(* Logix 5000 project; controller CLASE_1 Emulate 5570 rev 28.11; software revision 28.02; part 6 of 15 *)
(* tags used below, declared in another part *)
   Inp_RunFdbk : BOOL;   // Input Signal: RUN feedback from motor
   Inp_PermOK : BOOL;   // 1=Permissives OK, motor can start
   Inp_NBPermOK : BOOL;   // 1=Non-Bypassable Permissives OK, motor can start
   Inp_IntlkOK : BOOL;   // 1=Interlocks OK, motor can start/run
   Inp_NBIntlkOK : BOOL;   // 1=Non-Bypassable Interlocks OK, motor can start/run
   Inp_IOFault : BOOL;   // Input Communication Status 0=OK, 1=fail
   Inp_Sim : BOOL;   // 1=Simulate working motor; 0=Start/Stop/ Monitor actual motor
   Inp_OvrdCmd : DINT;   // Override Mode Command: 0=None, 1=Stop, 2=Start
   Cfg_HasRunFdbk : BOOL;   // 1=Motor provides run feedback
   Cfg_UseRunFdbk : BOOL;   // 1=Motor run feedback should be used for failure checking
   Cfg_AllowLocal : BOOL;   // 1=Allow Local Start/Stop without alarm, 0=Start/Stop from HMI/prog only
   Cfg_PCmdClear : ALIAS FOR Mode.Cfg_PCmdClear;
   Cfg_OperStopPrio : BOOL;   // 1=OCmd_Stop available in any mode, 0=OCmd_Stop only in Oper, Maint modes.
   Cfg_OCmdResets : BOOL;   // 1=New Oper motor cmd. resets fault, 0=reset req'd to clear fault
   Cfg_ShedOnFailToStart : BOOL;   // 1=Stop Motor and Alarm on Fail to Start; 0=Alarm only on Fail to Start
   Cfg_ShedOnIOFault : BOOL;   // 1=Stop Motor and Alarm on I/O Fault; 0=Alarm only on I/O Fault
   PCmd_Start : BOOL;   // Program Command to Start Motor
   PCmd_Stop : BOOL;   // Program Command to Stop Motor
   OCmd_Start : BOOL;   // Operator Command to Start Motor
   OCmd_Stop : BOOL;   // Operator Command to Stop Motor
   Out_Run : BOOL;   // 1=Run Motor, 0=Stop Motor
   Out_Start : BOOL;   // 1=Start Motor, 0=Motor left in current state
   Out_Stop : BOOL;   // 1=Stop Motor, 0=Motor left in current state
   SrcQ_IO : SINT;   // Source and Quality of primary I/O (enumeration)
   SrcQ : SINT;   // Source and Quality of primary Val/Sts (enumeration)
   Val_Cmd : SINT;   // Device Command 0=None, 1=Stop, 2=Start
   Val_Sts : SINT;   // Device Confirmed Sts 0=? 1=Stopped, 2=Running, 7=Stopping, 8=Starting, 33=Disabled
   Val_Fault : SINT;   // Device Fault Status 0=None, 16=Fail to Start, 17 = Fail to Stop, 32=I/O Fault, 34=Config Error
   Val_Notify : SINT;   // Current Alarm Level and Acknowledgement (enumeration)
   Sts_Stopped : BOOL;   // 1=Motor requested to stop and is confirmed stopped
   Sts_Starting : BOOL;   // 1=Motor requested to run and awaiting run feedback
   Sts_Running : BOOL;   // 1=Motor requested to run and is confirmed running
   Sts_Stopping : BOOL;   // 1=Motor requested to stop and awaiting stopped feedback
   Sts_Available : BOOL;   // 1=Motor available for control by automation (Prog)
   Sts_BypActive : BOOL;   // 1=Bypassing Active (Bypassed or Maintenance)
   Sts_Disabled : BOOL;   // 1=Motor is Disabled
   Sts_NotRdy : BOOL;   // 1=Device Not Ready, see detail bits for reason
   Nrdy_Disabled : BOOL;   // 1=Device Not Ready: Device Disabled by Maintenance
   Nrdy_CfgErr : BOOL;   // 1=Device Not Ready: Configuration Error
   Nrdy_Intlk : BOOL;   // 1=Device Not Ready: Interlock Not OK
   Nrdy_Perm : BOOL;   // 1=Device Not Ready: Permissive Not OK
   Nrdy_OperPrio : BOOL;   // 1=Device Not Ready: Operator State 0 Priority Command Requires Reset
   Nrdy_Fail : BOOL;   // 1=Device Not Ready: Device Failure (Shed Requires Reset)
   Nrdy_IOFault : BOOL;   // 1=Device Not Ready: I/O Fault (Shed Requires Reset)
   Nrdy_NoMode : BOOL;   // 1=Device Not Ready: Device Logic Disabled / NO Mode
   Sts_AlmInh : BOOL;   // 1=An Alarm is Shelved, Disabled or Suppressed: display icon
   Sts_Err : BOOL;   // 1=Error in Config: see detail bits for reason
   Sts_Hand : ALIAS FOR Mode.Sts_Hand;
   Sts_Maint : ALIAS FOR Mode.Sts_Maint;
   Sts_Ovrd : ALIAS FOR Mode.Sts_Ovrd;
   Sts_Prog : ALIAS FOR Mode.Sts_Prog;
   Sts_Oper : ALIAS FOR Mode.Sts_Oper;
   Sts_FailToStart : ALIAS FOR FailToStart.Inp;   // 1=Motor Failed to Start (one-shot)
   Sts_FailToStop : ALIAS FOR FailToStop.Inp;   // 1=Motor Failed to Stop
   Sts_IntlkTrip : ALIAS FOR IntlkTrip.Inp;   // 1=Motor stopped by an Interlock NOT OK (one-shot)
   Sts_IOFault : ALIAS FOR IOFault.Inp;   // I/O Comm Fault Status (0=OK, 1=Bad)
   Rdy_Start : BOOL;   // 1=Ready to receive OCmd_Start (enables HMI button)
   Rdy_Stop : BOOL;   // 1=Ready to receive OCmd_Stop (enables HMI button)
   Rdy_Reset : BOOL;   // 1=At least one Alarm or Latched Shed requires Reset
   Rdy_ResetAckAll : BOOL;   // 1=At least one Alarm or latched Shed condition requires Reset or Ack
   P_Motor : BOOL;   // Unique Parameter Name for auto - discovery
   Mode : P_Mode;   // Motor Mode Selection
   IOFault : P_Alarm;   // I/O Fault Alarm
   IntlkTrip : P_Alarm;   // Interlock Trip Alarm
   FailToStop : P_Alarm;   // Motor Failed to Stop Alarm
   FailToStart : P_Alarm;   // Motor Failed to Start Alarm
   Wrk_Run : BOOL;   // 1=Motor should be "running", 0=should be "stopped"
   Wrk_SimRunT : TIMER;   // Simulation Delay until Running
   Wrk_StopT : TIMER;   // Stop Check Timer
   Wrk_StartT : TIMER;   // Start Check Timer
   Wrk_SimStopT : TIMER;   // Simulation Delay until Stopped
   Wrk_RunFdbk : BOOL;   // Run Feedback based on mode, simulation, etc. 1=running
   Wrk_Notify : DINT;   // Buffer for building Val_Notify
   Wrk_Cmd : SINT;   // Buffer for building Val_Cmd
   Wrk_Sts : SINT;   // Buffer for building Val_Sts
   Wrk_Fault : SINT;   // Buffer for building Val_Fault
   Wrk_Retrigger : BOOL;   // Maint Start issued while running or Stop while stopped
   Wrk_SrcQ : SINT;   // Register for building Source / Quality enumeration
   Wrk_NotRdyONS : BOOL;   // Assert Stop on One-Shot of Sts_NotRdy
   Wrk_NotRdy : BOOL;   // Device Not Ready conditions excluding shed latches
   Wrk_StopInhT : TIMER;   // Local Stop Inhibit Timer
   Wrk_StartInhT : TIMER;   // Local Start Inhibit Timer
   Wrk_NoLongerSim : BOOL;   // Switched from Simulated to Real Motor this scan
(* P_Motor, continued *)

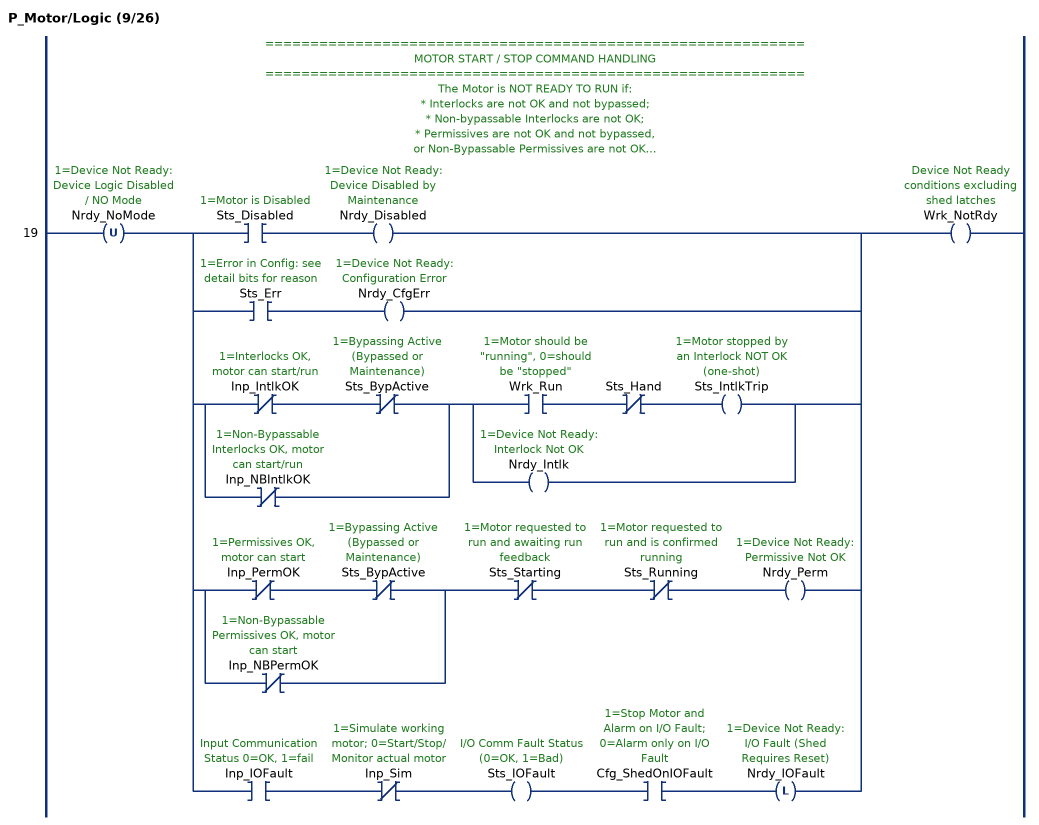
   // ============================================================
   // MOTOR START / STOP COMMAND HANDLING
   // ============================================================
   // The Motor is NOT READY TO RUN if:
   // * Interlocks are not OK and not bypassed;
   // * Non-bypassable Interlocks are not OK;
   // * Permissives are not OK and not bypassed,
   // or Non-Bypassable Permissives are not OK,
   // and the motor is not already starting or running;
   // * There's an I/O failure and the motor is NOT being simulated;
   // * The motor has a Fail to Start or Fail to Stop that has not been reset;
   // * The motor is disabled by Maintenance.
   // #####  V3.1-00  2014-06-30: Added Not Ready reason bits (Nrdy_xxx)  #####
   // #####  V3.1-01  2014-08-29:  Corrections to Nrdy_ trip and reset logic.  #####
   // #####  V3.5-09  2018-01-11:  Modified to ensure HAND running shows status RUNNING.  #####
   19: OTU(Nrdy_NoMode)[XIC(Sts_Disabled) OTE(Nrdy_Disabled) ,XIC(Sts_Err) OTE(Nrdy_CfgErr) ,[XIO(Inp_IntlkOK) XIO(Sts_BypActive) ,XIO(Inp_NBIntlkOK) ] [XIC(Wrk_Run) XIO(Sts_Hand) OTE(Sts_IntlkTrip) ,OTE(Nrdy_Intlk) ] ,[XIO(Inp_PermOK) XIO(Sts_BypActive) ,XIO(Inp_NBPermOK) ] XIO(Sts_Starting) XIO(Sts_Running) OTE(Nrdy_Perm) ,XIC(Inp_IOFault) XIO(Inp_Sim) OTE(Sts_IOFault) XIC(Cfg_ShedOnIOFault) OTL(Nrdy_IOFault) ]OTE(Wrk_NotRdy);
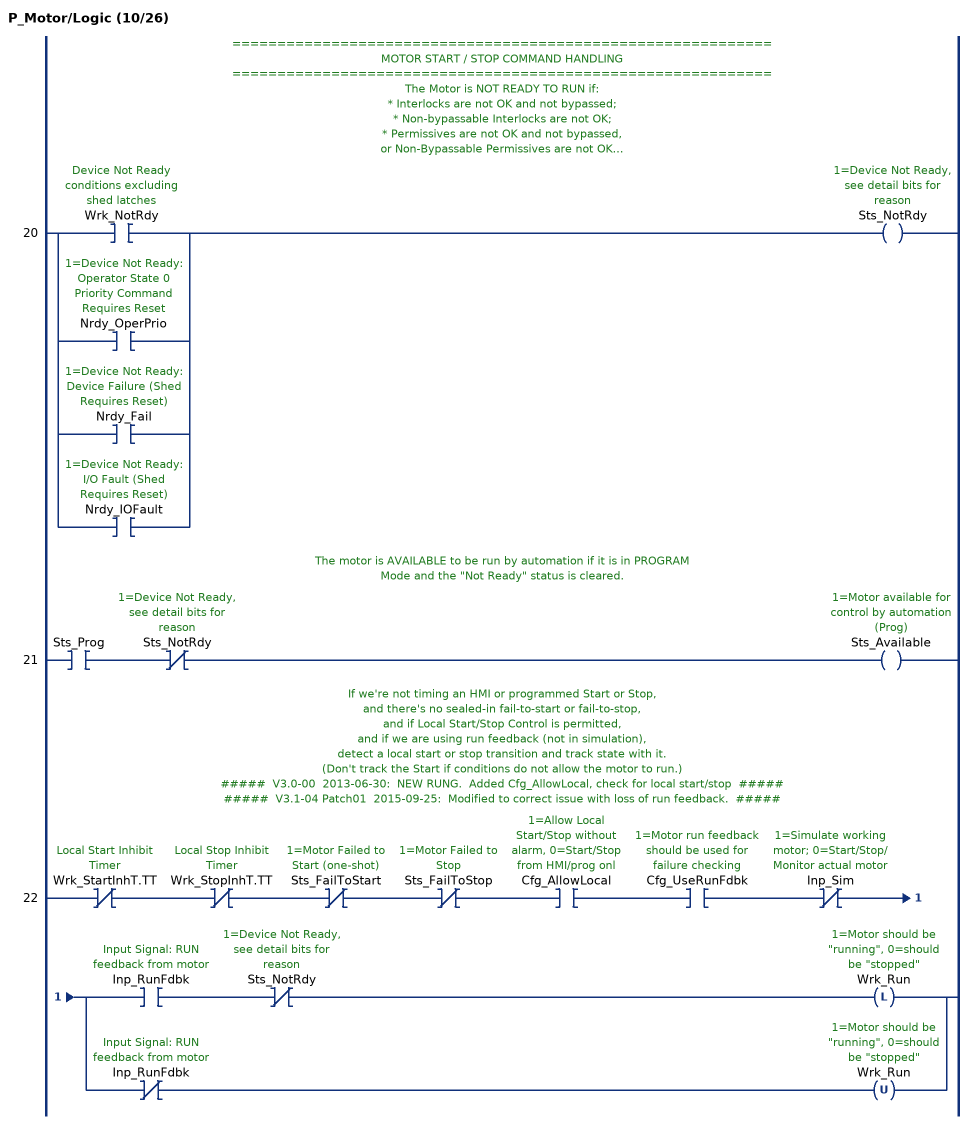
   // ============================================================
   // MOTOR START / STOP COMMAND HANDLING
   // ============================================================
   // The Motor is NOT READY TO RUN if:
   // * Interlocks are not OK and not bypassed;
   // * Non-bypassable Interlocks are not OK;
   // * Permissives are not OK and not bypassed,
   // or Non-Bypassable Permissives are not OK,
   // and the motor is not already starting or running;
   // * There's an I/O failure and the motor is NOT being simulated;
   // * The motor has a Fail to Start or Fail to Stop that has not been reset;
   // * The motor is disabled by Maintenance.
   // #####  V3.1-00  2014-06-30: Added Not Ready reason bits (Nrdy_xxx)  #####
   // #####  V3.1-01  2014-08-29:  Corrections to Nrdy_ trip and reset logic.  #####
   20: [XIC(Wrk_NotRdy) ,XIC(Nrdy_OperPrio) ,XIC(Nrdy_Fail) ,XIC(Nrdy_IOFault) ]OTE(Sts_NotRdy);
   // The motor is AVAILABLE to be run by automation if it is in PROGRAM
   // Mode and the "Not Ready" status is cleared.
   21: XIC(Sts_Prog)XIO(Sts_NotRdy)OTE(Sts_Available);
   // If we're not timing an HMI or programmed Start or Stop,
   // and there's no sealed-in fail-to-start or fail-to-stop,
   // and if Local Start/Stop Control is permitted,
   // and if we are using run feedback (not in simulation),
   // detect a local start or stop transition and track state with it.
   // (Don't track the Start if conditions do not allow the motor to run.)
   // #####  V3.0-00  2013-06-30:  NEW RUNG.  Added Cfg_AllowLocal, check for local start/stop  #####
   // #####  V3.1-04 Patch01  2015-09-25:  Modified to correct issue with loss of run feedback.  #####
   22: XIO(Wrk_StartInhT.TT)XIO(Wrk_StopInhT.TT)XIO(Sts_FailToStart)XIO(Sts_FailToStop)XIC(Cfg_AllowLocal)XIC(Cfg_UseRunFdbk)XIO(Inp_Sim)[XIC(Inp_RunFdbk) XIO(Sts_NotRdy) OTL(Wrk_Run) ,XIO(Inp_RunFdbk) OTU(Wrk_Run) ];
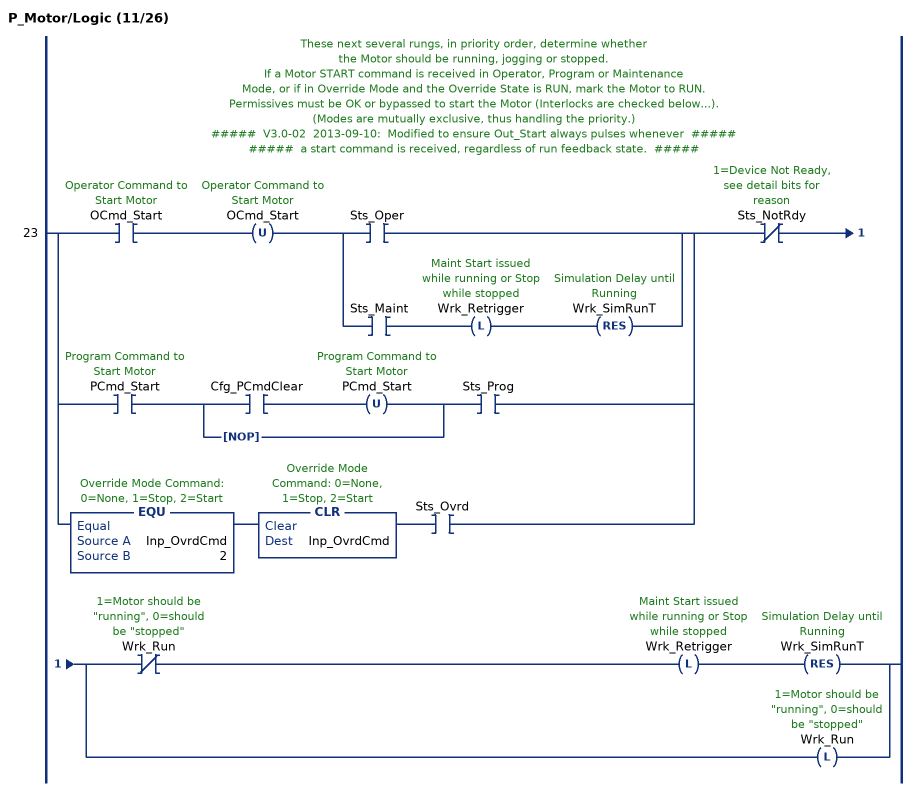
   // These next several rungs, in priority order, determine whether
   // the Motor should be running, jogging or stopped.
   // If a Motor START command is received in Operator, Program or Maintenance
   // Mode, or if in Override Mode and the Override State is RUN, mark the Motor to RUN.
   // Permissives must be OK or bypassed to start the Motor (Interlocks are checked below...).
   // (Modes are mutually exclusive, thus handling the priority.)
   // #####  V3.0-02  2013-09-10:  Modified to ensure Out_Start always pulses whenever  #####
   // #####  a start command is received, regardless of run feedback state.  #####
   23: [XIC(OCmd_Start) OTU(OCmd_Start) [XIC(Sts_Oper) ,XIC(Sts_Maint) OTL(Wrk_Retrigger) RES(Wrk_SimRunT) ] ,XIC(PCmd_Start) [XIC(Cfg_PCmdClear) OTU(PCmd_Start) ,NOP() ] XIC(Sts_Prog) ,EQU(Inp_OvrdCmd,2) CLR(Inp_OvrdCmd) XIC(Sts_Ovrd) ]XIO(Sts_NotRdy)[XIO(Wrk_Run) OTL(Wrk_Retrigger) RES(Wrk_SimRunT) ,OTL(Wrk_Run) ];
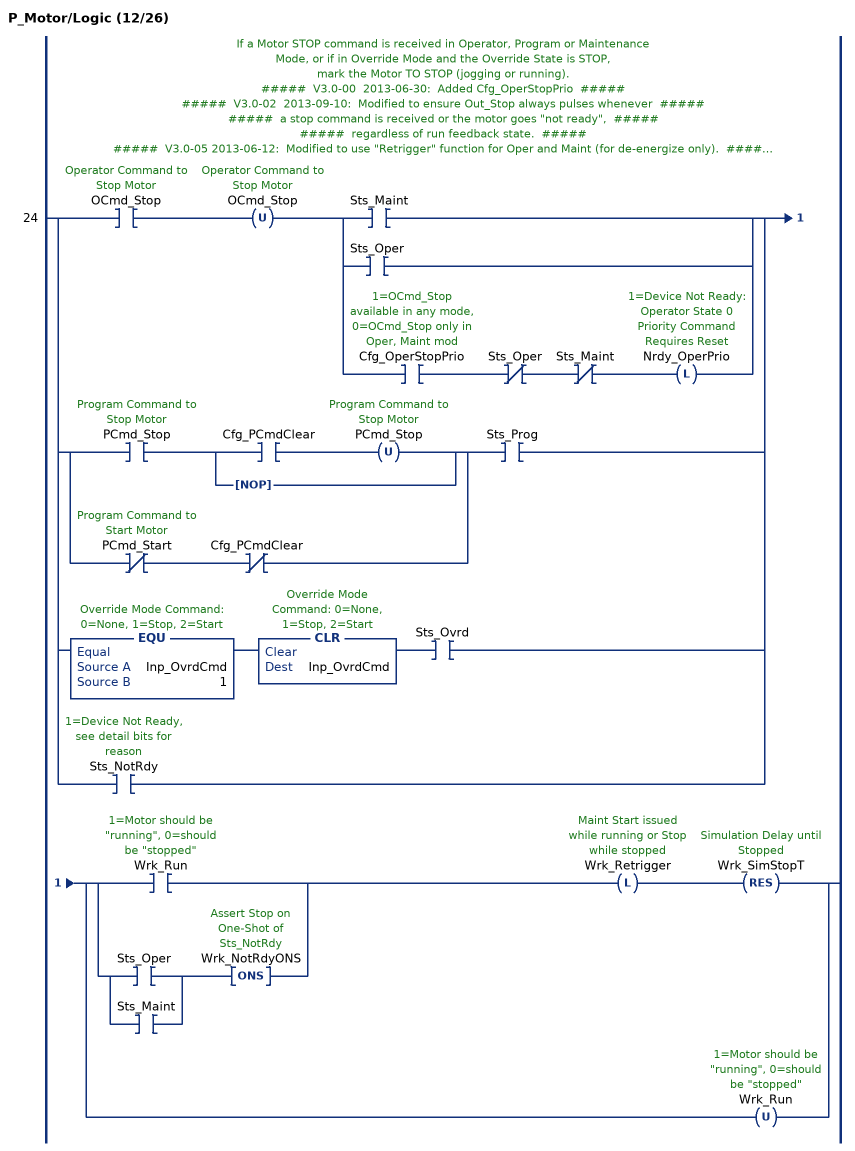
   // If a Motor STOP command is received in Operator, Program or Maintenance
   // Mode, or if in Override Mode and the Override State is STOP,
   // mark the Motor TO STOP (jogging or running).
   // #####  V3.0-00  2013-06-30:  Added Cfg_OperStopPrio  #####
   // #####  V3.0-02  2013-09-10:  Modified to ensure Out_Stop always pulses whenever  #####
   // #####  a stop command is received or the motor goes "not ready",  #####
   // #####  regardless of run feedback state.  #####
   // #####  V3.0-05 2013-06-12:  Modified to use "Retrigger" function for Oper and Maint (for de-energize only).  #####
   // #####  V3.1-00  2014-06-30: Added Not Ready reason bits (Nrdy_xxx)  #####
   // #####  V3.1-01 2014-08-29:  Resolved held "Stopping" status.  #####
   // #####  V3.1-03  2015-01-16:   Modified stop retriggering to handle asynchronous Prog mode owner.  #####
   24: [XIC(OCmd_Stop) OTU(OCmd_Stop) [[XIC(Sts_Maint) ,XIC(Sts_Oper) ] ,XIC(Cfg_OperStopPrio) XIO(Sts_Oper) XIO(Sts_Maint) OTL(Nrdy_OperPrio) ] ,[XIC(PCmd_Stop) [XIC(Cfg_PCmdClear) OTU(PCmd_Stop) ,NOP() ] ,XIO(PCmd_Start) XIO(Cfg_PCmdClear) ] XIC(Sts_Prog) ,EQU(Inp_OvrdCmd,1) CLR(Inp_OvrdCmd) XIC(Sts_Ovrd) ,XIC(Sts_NotRdy) ][[XIC(Wrk_Run) ,[XIC(Sts_Oper) ,XIC(Sts_Maint) ] ONS(Wrk_NotRdyONS) ] OTL(Wrk_Retrigger) RES(Wrk_SimStopT) ,OTU(Wrk_Run) ];
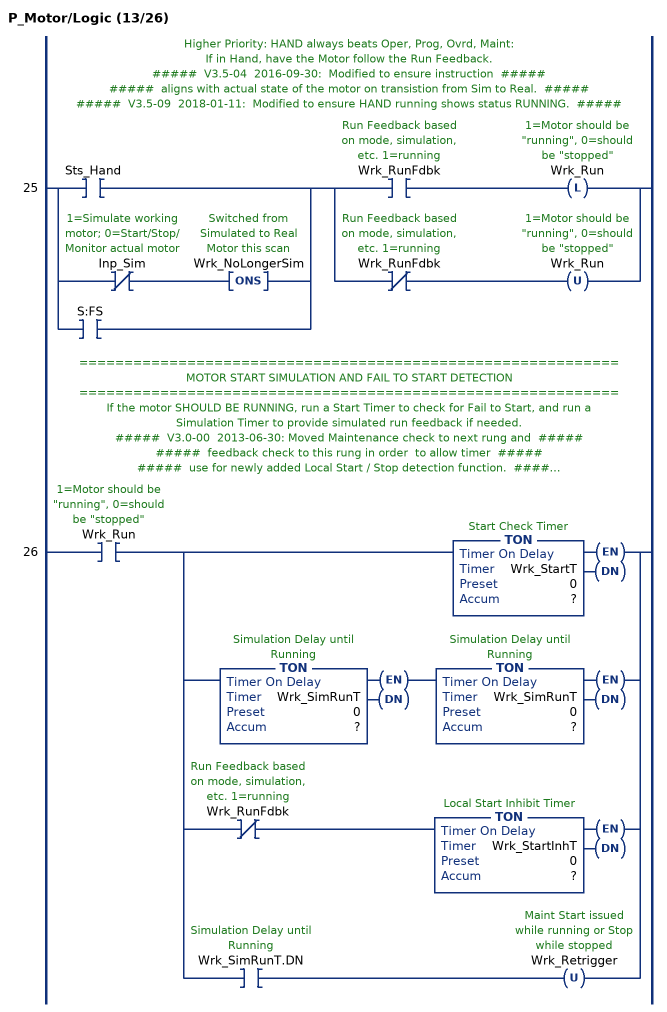
   // Higher Priority: HAND always beats Oper, Prog, Ovrd, Maint:
   // If in Hand, have the Motor follow the Run Feedback.
   // #####  V3.5-04  2016-09-30:  Modified to ensure instruction  #####
   // #####  aligns with actual state of the motor on transistion from Sim to Real.  #####
   // #####  V3.5-09  2018-01-11:  Modified to ensure HAND running shows status RUNNING.  #####
   25: [XIC(Sts_Hand) ,XIO(Inp_Sim) ONS(Wrk_NoLongerSim) ,XIC(S:FS) ][XIC(Wrk_RunFdbk) OTL(Wrk_Run) ,XIO(Wrk_RunFdbk) OTU(Wrk_Run) ];
   // ============================================================
   // MOTOR START SIMULATION AND FAIL TO START DETECTION
   // ============================================================
   // If the motor SHOULD BE RUNNING, run a Start Timer to check for Fail to Start, and run a
   // Simulation Timer to provide simulated run feedback if needed.
   // #####  V3.0-00  2013-06-30: Moved Maintenance check to next rung and  #####
   // #####  feedback check to this rung in order  to allow timer  #####
   // #####  use for newly added Local Start / Stop detection function.  #####
   // #####  V3.1-04 Patch01  2015-09-25:  Modified to correct issue with loss of run feedback.  #####
   // @@@@@  The TON on the second branch is doubled to ensure it goes  @@@@@
   // @@@@@  the same scan it is enabled if its preset is zero.  @@@@@
   26: XIC(Wrk_Run)[TON(Wrk_StartT,?,?) ,TON(Wrk_SimRunT,?,?) TON(Wrk_SimRunT,?,?) ,XIO(Wrk_RunFdbk) TON(Wrk_StartInhT,?,?) ,XIC(Wrk_SimRunT.DN) OTU(Wrk_Retrigger) ];
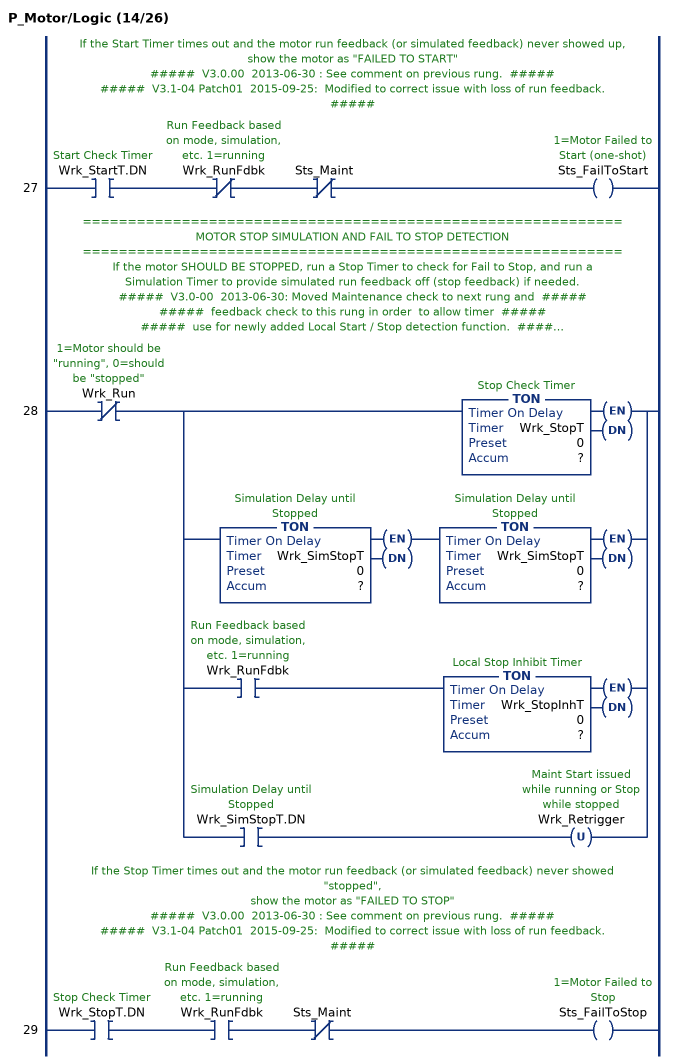
   // If the Start Timer times out and the motor run feedback (or simulated feedback) never showed up,
   // show the motor as "FAILED TO START"
   // #####  V3.0.00  2013-06-30 : See comment on previous rung.  #####
   // #####  V3.1-04 Patch01  2015-09-25:  Modified to correct issue with loss of run feedback.  #####
   27: XIC(Wrk_StartT.DN)XIO(Wrk_RunFdbk)XIO(Sts_Maint)OTE(Sts_FailToStart);
   // ============================================================
   // MOTOR STOP SIMULATION AND FAIL TO STOP DETECTION
   // ============================================================
   // If the motor SHOULD BE STOPPED, run a Stop Timer to check for Fail to Stop, and run a
   // Simulation Timer to provide simulated run feedback off (stop feedback) if needed.
   // #####  V3.0-00  2013-06-30: Moved Maintenance check to next rung and  #####
   // #####  feedback check to this rung in order  to allow timer  #####
   // #####  use for newly added Local Start / Stop detection function.  #####
   // #####  V3.1-04 Patch01  2015-09-25:  Modified to correct issue with loss of run feedback.  #####
   // @@@@@  The TON on the second branch is doubled to ensure it goes  @@@@@
   // @@@@@  the same scan it is enabled if its preset is zero.  @@@@@
   28: XIO(Wrk_Run)[TON(Wrk_StopT,?,?) ,TON(Wrk_SimStopT,?,?) TON(Wrk_SimStopT,?,?) ,XIC(Wrk_RunFdbk) TON(Wrk_StopInhT,?,?) ,XIC(Wrk_SimStopT.DN) OTU(Wrk_Retrigger) ];
   // If the Stop Timer times out and the motor run feedback (or simulated feedback) never showed "stopped",
   // show the motor as "FAILED TO STOP"
   // #####  V3.0.00  2013-06-30 : See comment on previous rung.  #####
   // #####  V3.1-04 Patch01  2015-09-25:  Modified to correct issue with loss of run feedback.  #####
   29: XIC(Wrk_StopT.DN)XIC(Wrk_RunFdbk)XIO(Sts_Maint)OTE(Sts_FailToStop);
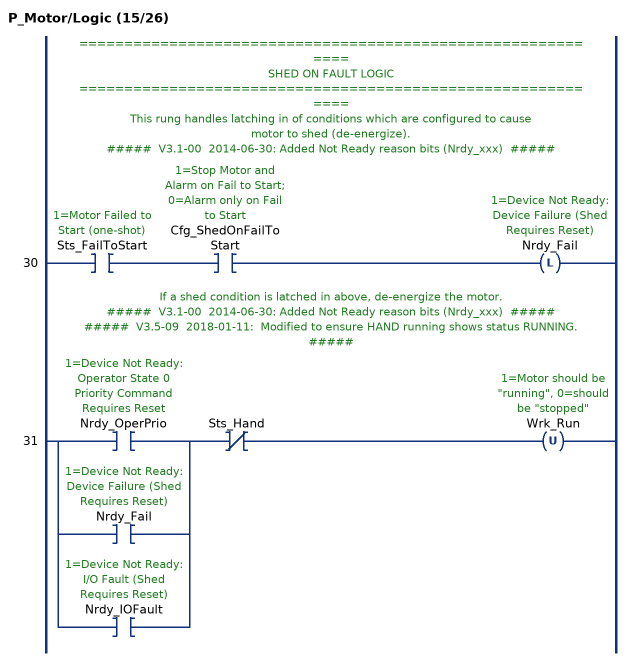
   // ============================================================
   // SHED ON FAULT LOGIC
   // ============================================================
   // This rung handles latching in of conditions which are configured to cause
   // motor to shed (de-energize).
   // #####  V3.1-00  2014-06-30: Added Not Ready reason bits (Nrdy_xxx)  #####
   30: XIC(Sts_FailToStart)XIC(Cfg_ShedOnFailToStart)OTL(Nrdy_Fail);
   // If a shed condition is latched in above, de-energize the motor.
   // #####  V3.1-00  2014-06-30: Added Not Ready reason bits (Nrdy_xxx)  #####
   // #####  V3.5-09  2018-01-11:  Modified to ensure HAND running shows status RUNNING.  #####
   31: [XIC(Nrdy_OperPrio) ,XIC(Nrdy_Fail) ,XIC(Nrdy_IOFault) ]XIO(Sts_Hand)OTU(Wrk_Run);
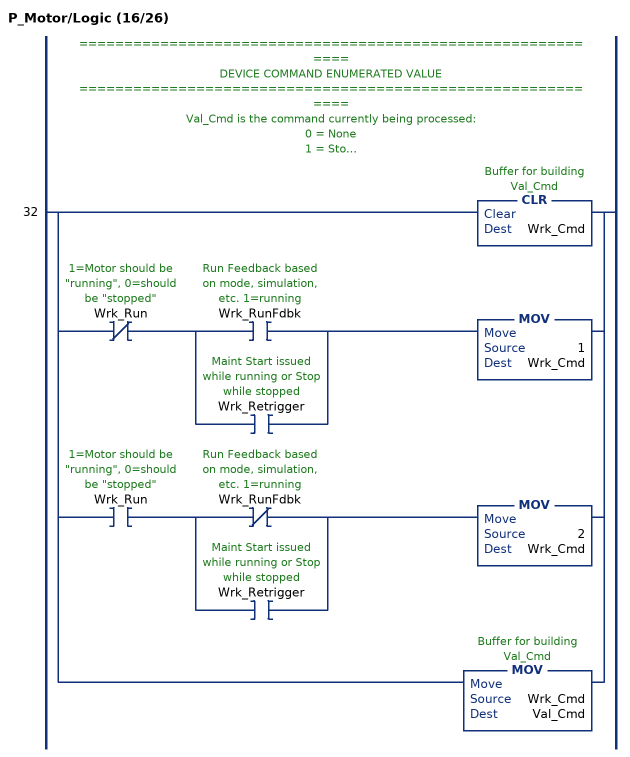
   // ============================================================
   // DEVICE COMMAND ENUMERATED VALUE
   // ============================================================
   // Val_Cmd is the command currently being processed:
   // 0 = None
   // 1 = Stop
   // 2 = Start
   32: [CLR(Wrk_Cmd) ,XIO(Wrk_Run) [XIC(Wrk_RunFdbk) ,XIC(Wrk_Retrigger) ] MOV(1,Wrk_Cmd) ,XIC(Wrk_Run) [XIO(Wrk_RunFdbk) ,XIC(Wrk_Retrigger) ] MOV(2,Wrk_Cmd) ,MOV(Wrk_Cmd,Val_Cmd) ];
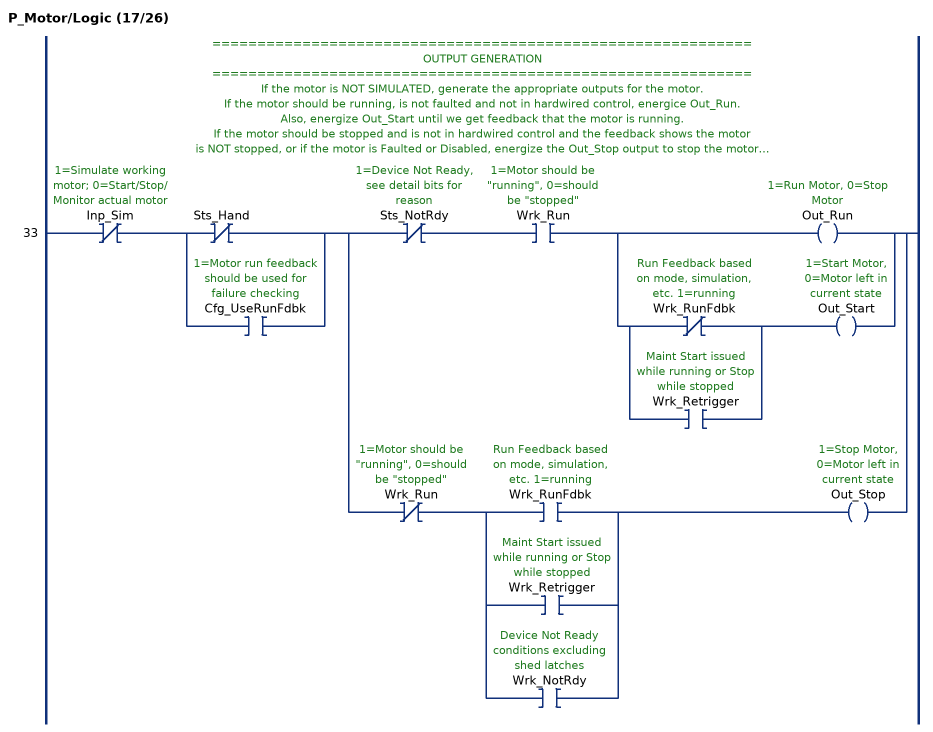
   // ============================================================
   // OUTPUT GENERATION
   // ============================================================
   // If the motor is NOT SIMULATED, generate the appropriate outputs for the motor.
   // If the motor should be running, is not faulted and not in hardwired control, energice Out_Run.
   // Also, energize Out_Start until we get feedback that the motor is running.
   // If the motor should be stopped and is not in hardwired control and the feedback shows the motor
   // is NOT stopped, or if the motor is Faulted or Disabled, energize the Out_Stop output to stop the motor.
   // #####  V3.0-05  2014-06-12:  Modified to energize Out_Stop on Shed conditions.  #####
   // #####  V3.1-00  2014-06-30: Added Not Ready reason bits (Nrdy_xxx)  #####
   33: XIO(Inp_Sim)[XIO(Sts_Hand) ,XIC(Cfg_UseRunFdbk) ][XIO(Sts_NotRdy) XIC(Wrk_Run) [OTE(Out_Run) ,[XIO(Wrk_RunFdbk) ,XIC(Wrk_Retrigger) ] OTE(Out_Start) ] ,XIO(Wrk_Run) [XIC(Wrk_RunFdbk) ,XIC(Wrk_Retrigger) ,XIC(Wrk_NotRdy) ] OTE(Out_Stop) ];
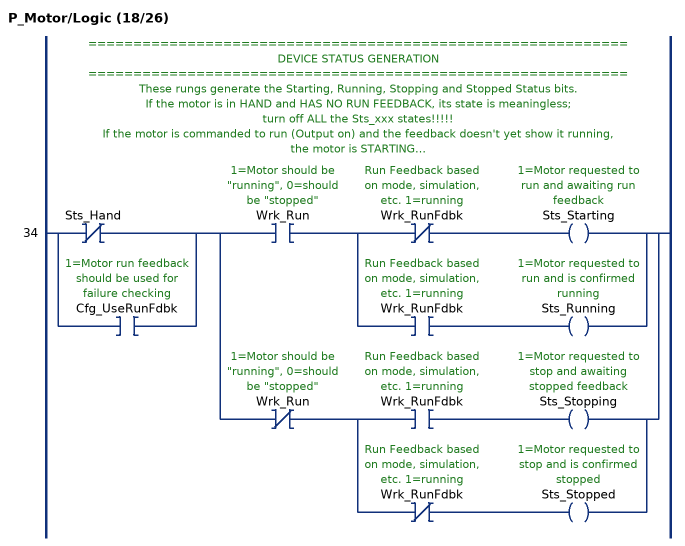
   // ============================================================
   // DEVICE STATUS GENERATION
   // ============================================================
   // These rungs generate the Starting, Running, Stopping and Stopped Status bits.
   // If the motor is in HAND and HAS NO RUN FEEDBACK, its state is meaningless;
   // turn off ALL the Sts_xxx states!!!!!
   // If the motor is commanded to run (Output on) and the feedback doesn't yet show it running,
   // the motor is STARTING.
   // If the motor is commanded to run (Output on) and the feedback shows it running,
   // the motor is RUNNING.
   // If the motor is commanded to stoop (Output off) and the feedback still shows it running,
   // the motor is STOPPING.
   // If the motor is commanded to stop (Output off) and the feedback shows it has stopped,
   // the motor is STOPPED.
   34: [XIO(Sts_Hand) ,XIC(Cfg_UseRunFdbk) ][XIC(Wrk_Run) [XIO(Wrk_RunFdbk) OTE(Sts_Starting) ,XIC(Wrk_RunFdbk) OTE(Sts_Running) ] ,XIO(Wrk_Run) [XIC(Wrk_RunFdbk) OTE(Sts_Stopping) ,XIO(Wrk_RunFdbk) OTE(Sts_Stopped) ] ];
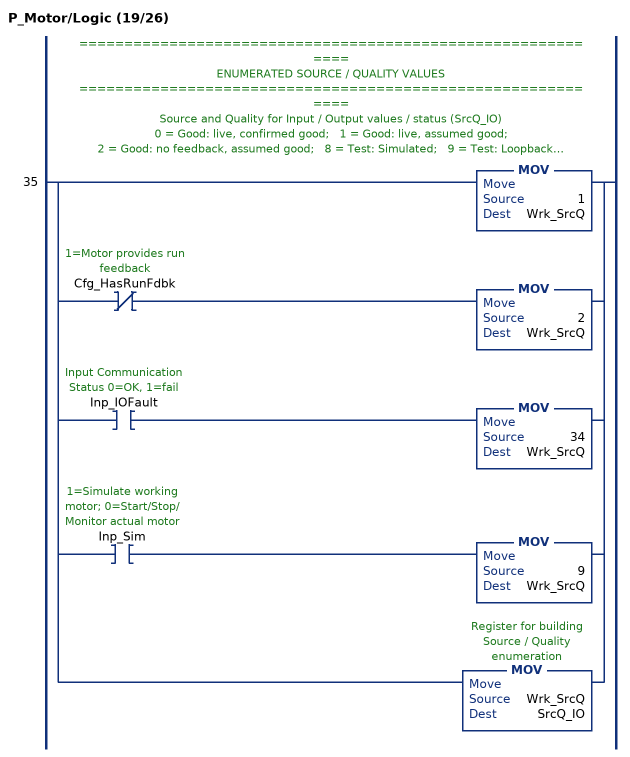
   // ============================================================
   // ENUMERATED SOURCE / QUALITY VALUES
   // ============================================================
   // Source and Quality for Input / Output values / status (SrcQ_IO)
   // 0 = Good: live, confirmed good;   1 = Good: live, assumed good;
   // 2 = Good: no feedback, assumed good;   8 = Test: Simulated;   9 = Test: Loopback;
   // 10 = Test: Manually Entered;   16 = Uncertain: Live, off-spec;
   // 17 = Uncertain, Substituted at Device / Bus;   18 = Uncertain, Substituted at AOI;
   // 19 = Uncertain, using last known good;    20 = Uncertain, using replacement value;
   // 32 = Bad, Signal Failure;   33 = Bad, Channel Fault;
   // 34 = Bad, Module / Comms Fault;   35 = Bad, Invalid Configuration
   // #####  V3.1-00  2014-06-30:  Added rung for Source/Quality enumerations.  #####
   35: [MOV(1,Wrk_SrcQ) ,XIO(Cfg_HasRunFdbk) MOV(2,Wrk_SrcQ) ,XIC(Inp_IOFault) MOV(34,Wrk_SrcQ) ,XIC(Inp_Sim) MOV(9,Wrk_SrcQ) ,MOV(Wrk_SrcQ,SrcQ_IO) ];
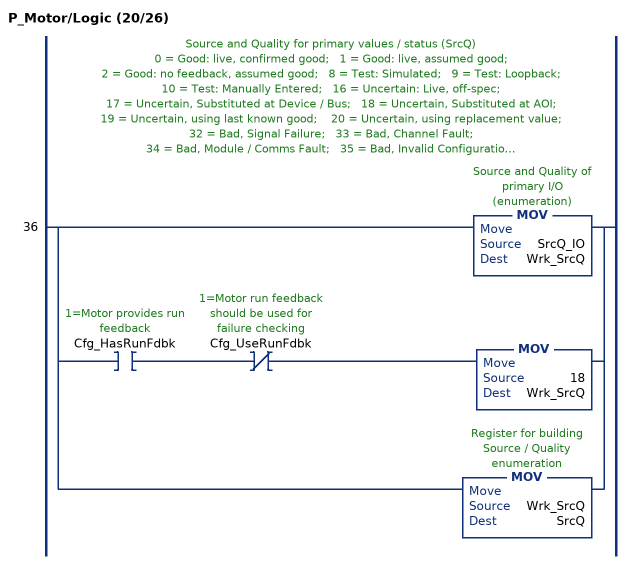
   // Source and Quality for primary values / status (SrcQ)
   // 0 = Good: live, confirmed good;   1 = Good: live, assumed good;
   // 2 = Good: no feedback, assumed good;   8 = Test: Simulated;   9 = Test: Loopback;
   // 10 = Test: Manually Entered;   16 = Uncertain: Live, off-spec;
   // 17 = Uncertain, Substituted at Device / Bus;   18 = Uncertain, Substituted at AOI;
   // 19 = Uncertain, using last known good;    20 = Uncertain, using replacement value;
   // 32 = Bad, Signal Failure;   33 = Bad, Channel Fault;
   // 34 = Bad, Module / Comms Fault;   35 = Bad, Invalid Configuration
   // #####  V3.1-00  2014-06-30:  Added rung for Source/Quality enumerations.  #####
   36: [MOV(SrcQ_IO,Wrk_SrcQ) ,XIC(Cfg_HasRunFdbk) XIO(Cfg_UseRunFdbk) MOV(18,Wrk_SrcQ) ,MOV(Wrk_SrcQ,SrcQ) ];
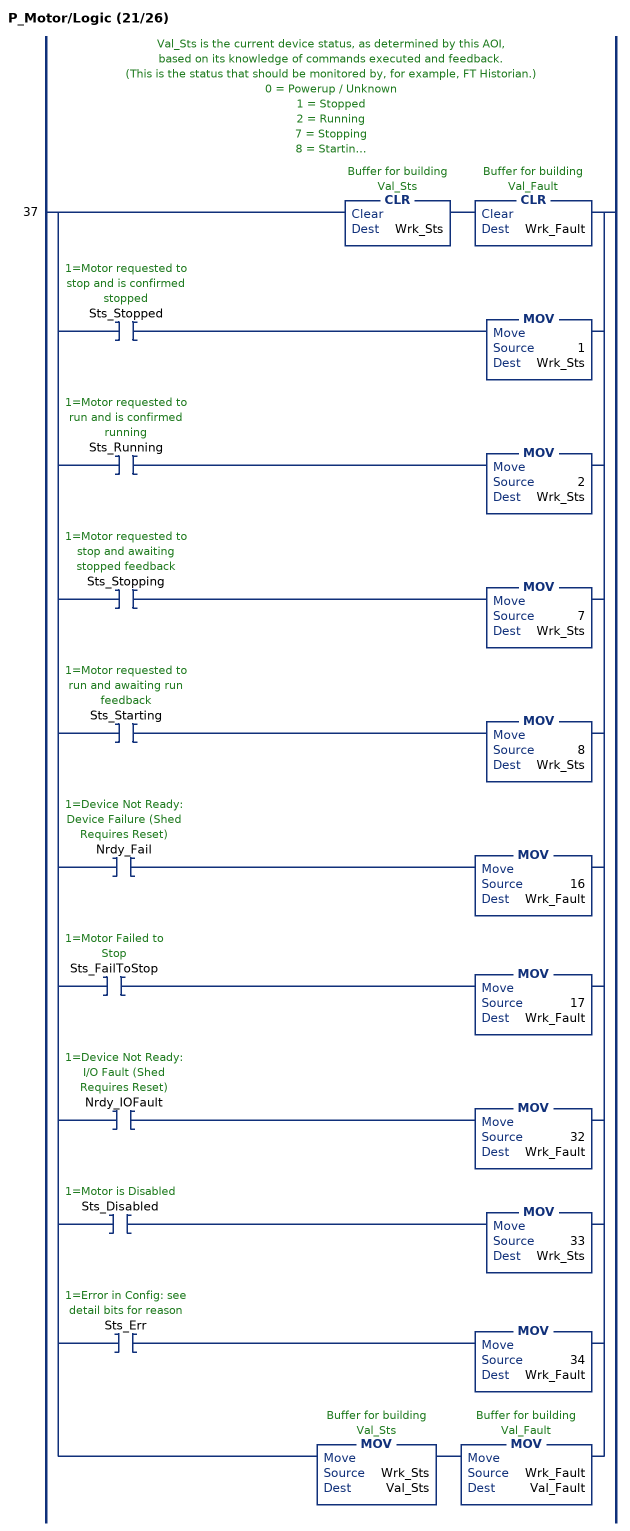
   // Val_Sts is the current device status, as determined by this AOI,
   // based on its knowledge of commands executed and feedback.
   // (This is the status that should be monitored by, for example, FT Historian.)
   // 0 = Powerup / Unknown
   // 1 = Stopped
   // 2 = Running
   // 7 = Stopping
   // 8 = Starting
   // 33 = Device Disabled
   // Val_Fault is the current device fault status, as determined by this AOI,
   // based on its knowledge of commands executed and feedback.
   // (This is the fault status that should be monitored by, for example, FT Historian.)
   // 0 = None
   // 16 = Fail to Start
   // 17 = Fail to Stop
   // 32 = I/O Fault (from Input)
   // 34 = Configuration Error
   // #####  V3.1-00  2014-06-30: Added Not Ready reason bits (Nrdy_xxx)  #####
   37: [CLR(Wrk_Sts) CLR(Wrk_Fault) ,XIC(Sts_Stopped) MOV(1,Wrk_Sts) ,XIC(Sts_Running) MOV(2,Wrk_Sts) ,XIC(Sts_Stopping) MOV(7,Wrk_Sts) ,XIC(Sts_Starting) MOV(8,Wrk_Sts) ,XIC(Nrdy_Fail) MOV(16,Wrk_Fault) ,XIC(Sts_FailToStop) MOV(17,Wrk_Fault) ,XIC(Nrdy_IOFault) MOV(32,Wrk_Fault) ,XIC(Sts_Disabled) MOV(33,Wrk_Sts) ,XIC(Sts_Err) MOV(34,Wrk_Fault) ,MOV(Wrk_Sts,Val_Sts) MOV(Wrk_Fault,Val_Fault) ];
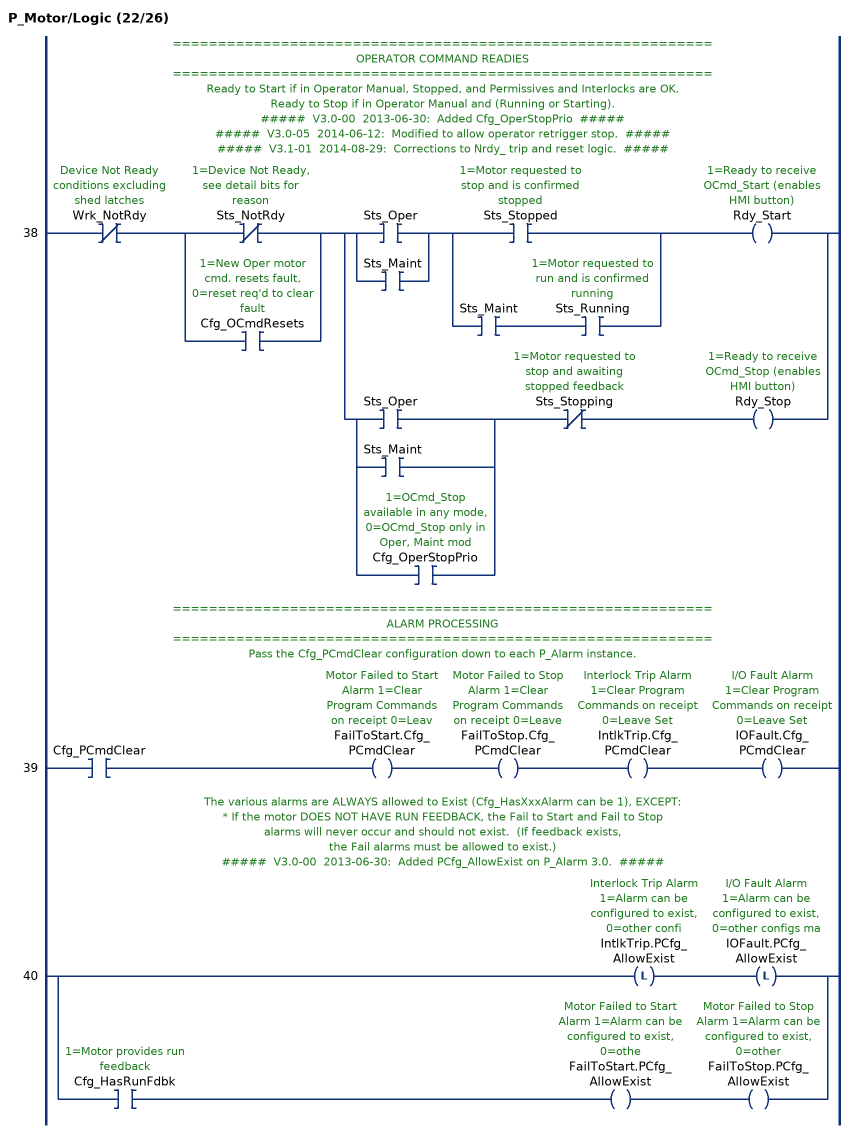
   // ============================================================
   // OPERATOR COMMAND READIES
   // ============================================================
   // Ready to Start if in Operator Manual, Stopped, and Permissives and Interlocks are OK.
   // Ready to Stop if in Operator Manual and (Running or Starting).
   // #####  V3.0-00  2013-06-30:  Added Cfg_OperStopPrio  #####
   // #####  V3.0-05  2014-06-12:  Modified to allow operator retrigger stop.  #####
   // #####  V3.1-01  2014-08-29:  Corrections to Nrdy_ trip and reset logic.  #####
   38: XIO(Wrk_NotRdy)[XIO(Sts_NotRdy) ,XIC(Cfg_OCmdResets) ][[XIC(Sts_Oper) ,XIC(Sts_Maint) ] [XIC(Sts_Stopped) ,XIC(Sts_Maint) XIC(Sts_Running) ] OTE(Rdy_Start) ,[XIC(Sts_Oper) ,XIC(Sts_Maint) ,XIC(Cfg_OperStopPrio) ] XIO(Sts_Stopping) OTE(Rdy_Stop) ];
   // ============================================================
   // ALARM PROCESSING
   // ============================================================
   // Pass the Cfg_PCmdClear configuration down to each P_Alarm instance.
   39: XIC(Cfg_PCmdClear)OTE(FailToStart.Cfg_PCmdClear)OTE(FailToStop.Cfg_PCmdClear)OTE(IntlkTrip.Cfg_PCmdClear)OTE(IOFault.Cfg_PCmdClear);
   // The various alarms are ALWAYS allowed to Exist (Cfg_HasXxxAlarm can be 1), EXCEPT:
   // * If the motor DOES NOT HAVE RUN FEEDBACK, the Fail to Start and Fail to Stop
   // alarms will never occur and should not exist.  (If feedback exists,
   // the Fail alarms must be allowed to exist.)
   // #####  V3.0-00  2013-06-30:  Added PCfg_AllowExist on P_Alarm 3.0.  #####
   40: [OTL(IntlkTrip.PCfg_AllowExist) OTL(IOFault.PCfg_AllowExist) ,XIC(Cfg_HasRunFdbk) OTE(FailToStart.PCfg_AllowExist) OTE(FailToStop.PCfg_AllowExist) ];
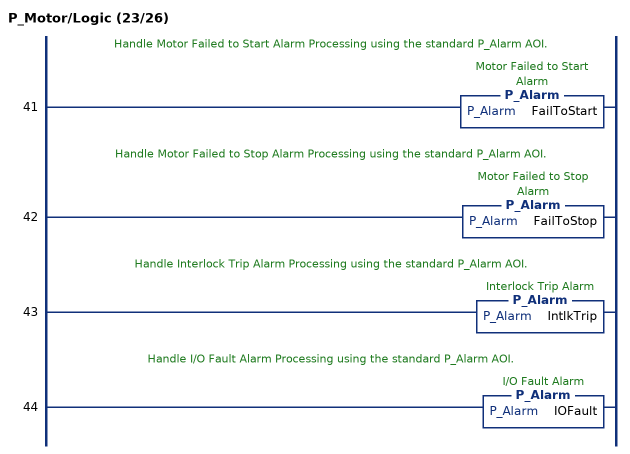
   // Handle Motor Failed to Start Alarm Processing using the standard P_Alarm AOI.
   41: P_Alarm(FailToStart);
   // Handle Motor Failed to Stop Alarm Processing using the standard P_Alarm AOI.
   42: P_Alarm(FailToStop);
   // Handle Interlock Trip Alarm Processing using the standard P_Alarm AOI.
   43: P_Alarm(IntlkTrip);
   // Handle I/O Fault Alarm Processing using the standard P_Alarm AOI.
   44: P_Alarm(IOFault);
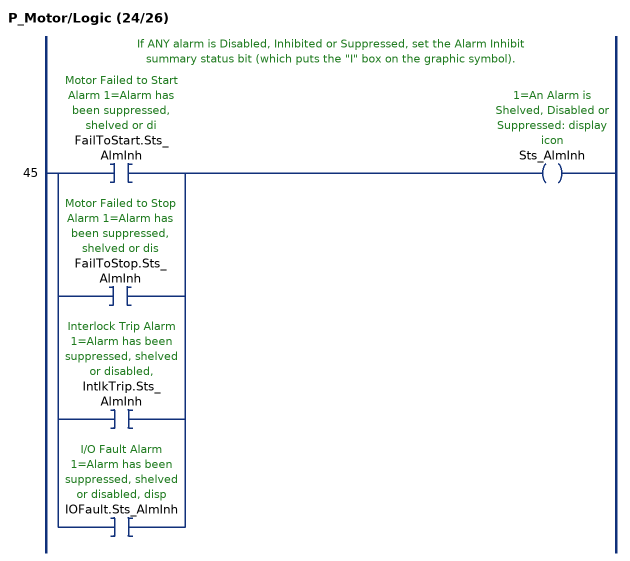
   // If ANY alarm is Disabled, Inhibited or Suppressed, set the Alarm Inhibit
   // summary status bit (which puts the "I" box on the graphic symbol).
   45: [XIC(FailToStart.Sts_AlmInh) ,XIC(FailToStop.Sts_AlmInh) ,XIC(IntlkTrip.Sts_AlmInh) ,XIC(IOFault.Sts_AlmInh) ]OTE(Sts_AlmInh);
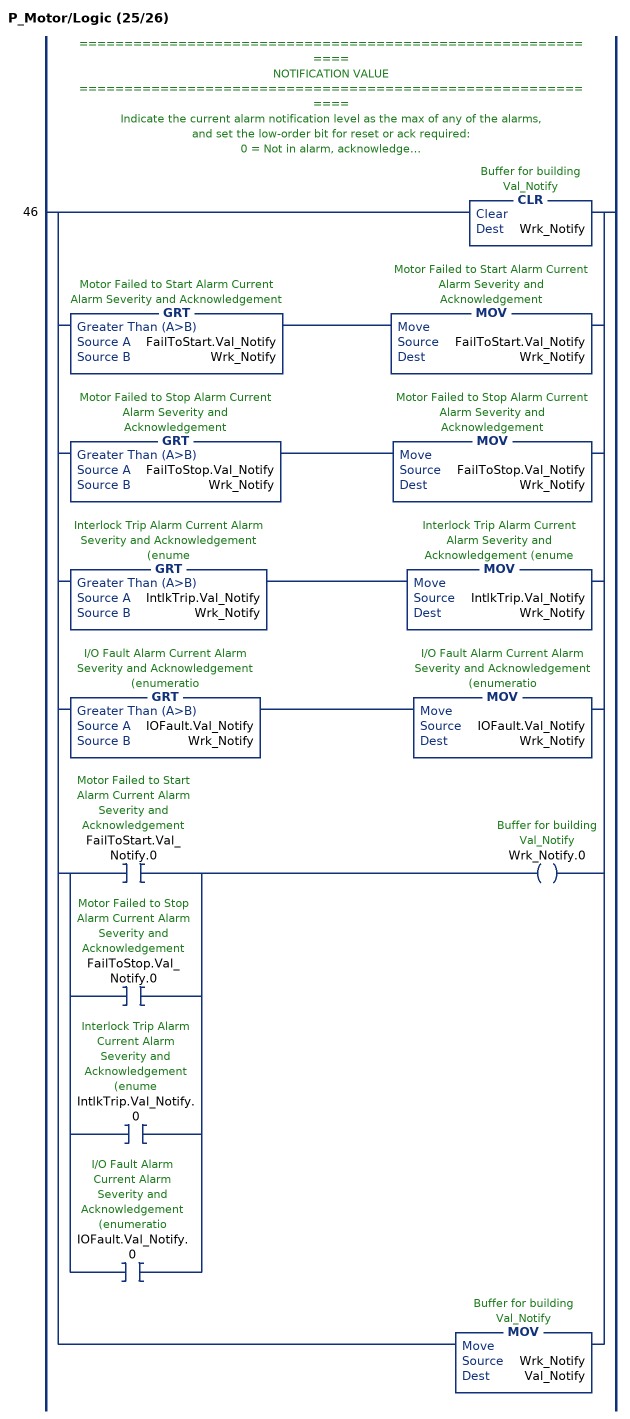
   // ============================================================
   // NOTIFICATION VALUE
   // ============================================================
   // Indicate the current alarm notification level as the max of any of the alarms,
   // and set the low-order bit for reset or ack required:
   // 0 = Not in alarm, acknowledged
   // 1 = Not in alarm, unacknowledged or reset required
   // 2 = Low severity alarm, acknowledged
   // 3 = Low severity alarm, unacknowledged
   // 4 = Medium severity alarm, acknowledged
   // 5 = Medium severity alarm, unacknowledged
   // 6 = High severity alarm, acknowledged
   // 7 = High severity alarm, unacknowledged
   // 8 = Urgent severity alarm, acknowledged
   // 9 = Urgent severity alarm, unacknowledged
   // #####  V3.1-00  2014-06-30:  Separated Reset Reqd functions from Val_Notify  #####
   46: [CLR(Wrk_Notify) ,GRT(FailToStart.Val_Notify,Wrk_Notify) MOV(FailToStart.Val_Notify,Wrk_Notify) ,GRT(FailToStop.Val_Notify,Wrk_Notify) MOV(FailToStop.Val_Notify,Wrk_Notify) ,GRT(IntlkTrip.Val_Notify,Wrk_Notify) MOV(IntlkTrip.Val_Notify,Wrk_Notify) ,GRT(IOFault.Val_Notify,Wrk_Notify) MOV(IOFault.Val_Notify,Wrk_Notify) ,[XIC(FailToStart.Val_Notify.0) ,XIC(FailToStop.Val_Notify.0) ,XIC(IntlkTrip.Val_Notify.0) ,XIC(IOFault.Val_Notify.0) ] OTE(Wrk_Notify.0) ,MOV(Wrk_Notify,Val_Notify) ];
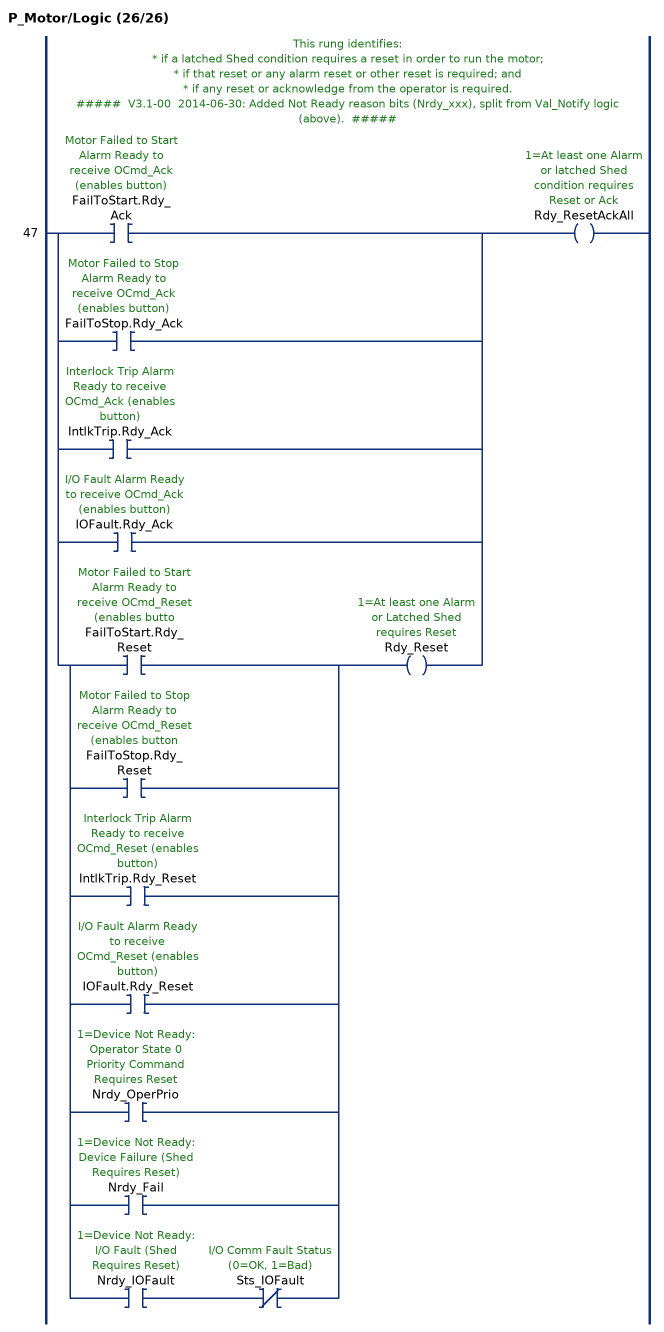
   // This rung identifies:
   // * if a latched Shed condition requires a reset in order to run the motor;
   // * if that reset or any alarm reset or other reset is required; and
   // * if any reset or acknowledge from the operator is required.
   // #####  V3.1-00  2014-06-30: Added Not Ready reason bits (Nrdy_xxx), split from Val_Notify logic (above).  #####
   47: [[XIC(FailToStart.Rdy_Ack) ,XIC(FailToStop.Rdy_Ack) ,XIC(IntlkTrip.Rdy_Ack) ,XIC(IOFault.Rdy_Ack) ] ,[XIC(FailToStart.Rdy_Reset) ,XIC(FailToStop.Rdy_Reset) ,XIC(IntlkTrip.Rdy_Reset) ,XIC(IOFault.Rdy_Reset) ,XIC(Nrdy_OperPrio) ,XIC(Nrdy_Fail) ,XIC(Nrdy_IOFault) XIO(Sts_IOFault) ] OTE(Rdy_Reset) ]OTE(Rdy_ResetAckAll);
END_ROUTINE
